// TIA Portal V17 export
// export: Created 2022-02-08T17:35:46.0434101Z, ExportSetting WithDefaults, DisplayName Totally Integrated Automation Portal, DisplayVersion V17 Update 2, DisplayName TIA Portal Openness, DisplayVersion V17 Update 2, DisplayName TIA Portal Version Control Interface, DisplayVersion V17, DisplayName STEP 7 Professional, DisplayVersion V17 Update 2, DisplayName STEP 7 Safety, DisplayVersion V17, DisplayName WinCC UA Professional, DisplayVersion V17 Update 2
FUNCTION_BLOCK "Motor"   // FB2, FBD
TITLE = Control module: Motor
{ S7_Optimized_Access := 'TRUE' }
VERSION : 0.1
// stored: AutoNumber true, IsIECCheckEnabled false, IsRetainMemResEnabled false, MemoryReserve 100, SetENOAutomatically false, UDAEnableTagReadback false
   VAR_INPUT
      i_Thermal : Bool;
      i_Mainswitch : Bool;
      i_SpareAlarm1 : Bool;
      i_SpareAlarm2 : Bool;
      i_SpareAlarm3 : Bool;
      i_SpareAlarm4 : Bool;
      i_InterlockDir1 : Bool;
      i_InterlockDir2 : Bool;
      i_EndswitchDir1 : Bool;
      i_EndswitchDir2 : Bool;
   END_VAR
   VAR_OUTPUT
      q_Dir1 : Bool;
      q_Dir2 : Bool;
      q_HighSpeed : Bool;
   END_VAR
   VAR_IN_OUT
      PLC_CtrlMod : "PLC_CtrlMod";
      HMI_CtrlMod : "HMI_CtrlMod";
   END_VAR
   VAR
      s_ManualMode : Bool;
      s_AutomaticMode : Bool;
      s_Direction1 : Bool;
      s_Direction2 : Bool;
      s_Alarms : Struct
         ThermalFaults : Bool;
         MainswitchOff : Bool;
         SpareAlarm1 : Bool;
         SpareAlarm2 : Bool;
         SpareAlarm3 : Bool;
         SpareAlarm4 : Bool;
      END_STRUCT;
   END_VAR
BEGIN

REGION Network 1: Selection manual mode
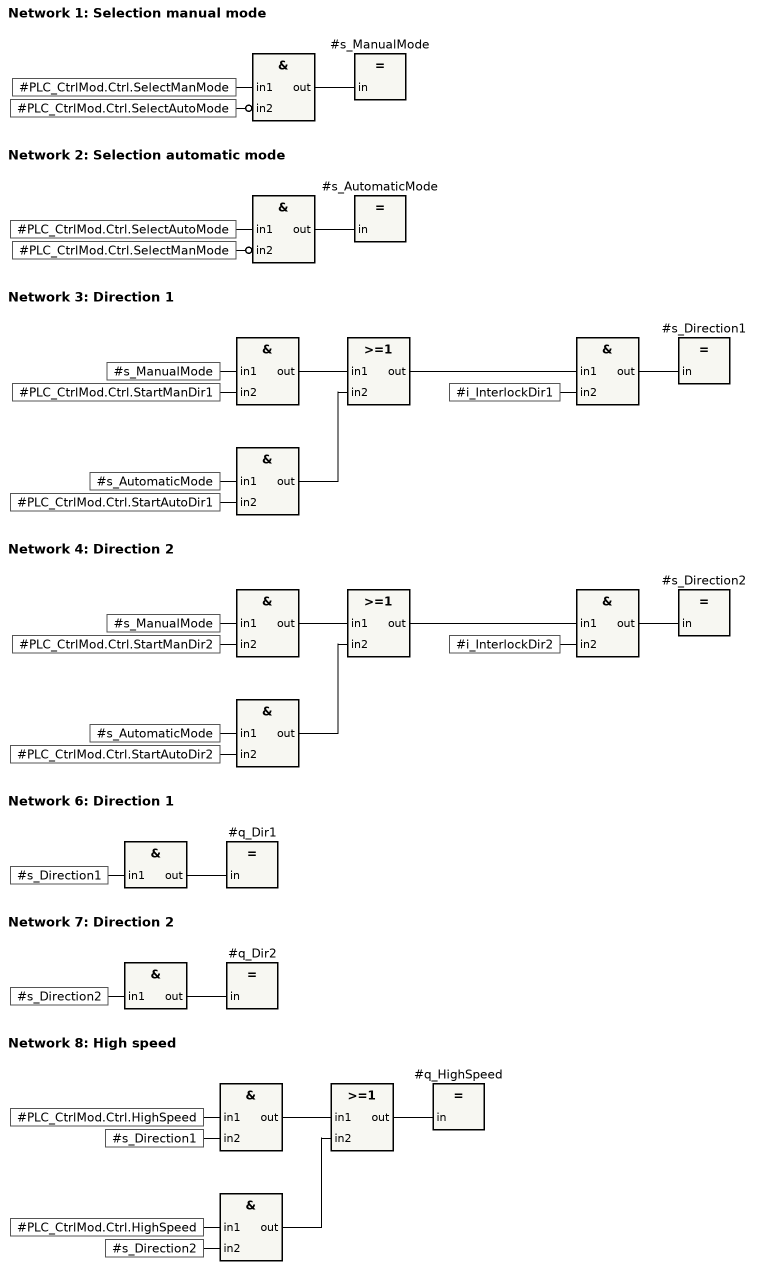
   #s_ManualMode := #PLC_CtrlMod.Ctrl.SelectManMode AND NOT #PLC_CtrlMod.Ctrl.SelectAutoMode;
END_REGION

REGION Network 2: Selection automatic mode
   #s_AutomaticMode := #PLC_CtrlMod.Ctrl.SelectAutoMode AND NOT #PLC_CtrlMod.Ctrl.SelectManMode;
END_REGION

REGION Network 3: Direction 1
   #s_Direction1 := ((#s_ManualMode AND #PLC_CtrlMod.Ctrl.StartManDir1) OR (#s_AutomaticMode AND #PLC_CtrlMod.Ctrl.StartAutoDir1)) AND #i_InterlockDir1;
END_REGION

REGION Network 4: Direction 2
   #s_Direction2 := ((#s_ManualMode AND #PLC_CtrlMod.Ctrl.StartManDir2) OR (#s_AutomaticMode AND #PLC_CtrlMod.Ctrl.StartAutoDir2)) AND #i_InterlockDir2;
END_REGION

REGION Network 5: ********* OUTPUTS *********
END_REGION

REGION Network 6: Direction 1
   #q_Dir1 := #s_Direction1;
END_REGION

REGION Network 7: Direction 2
   #q_Dir2 := #s_Direction2;
END_REGION

REGION Network 8: High speed
   #q_HighSpeed := (#PLC_CtrlMod.Ctrl.HighSpeed AND #s_Direction1) OR (#PLC_CtrlMod.Ctrl.HighSpeed AND #s_Direction2);
END_REGION

REGION Network 9: ********* ALARMS *********
END_REGION

REGION Network 10: Thermal fault
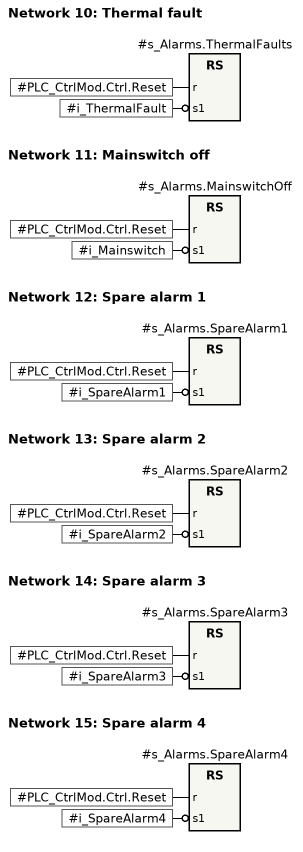
   IF #PLC_CtrlMod.Ctrl.Reset THEN
       #s_Alarms.ThermalFaults := FALSE;   // RS flip-flop
   END_IF;
   IF NOT #i_ThermalFault THEN #s_Alarms.ThermalFaults := TRUE; END_IF;
END_REGION

REGION Network 11: Mainswitch off
   IF #PLC_CtrlMod.Ctrl.Reset THEN
       #s_Alarms.MainswitchOff := FALSE;   // RS flip-flop
   END_IF;
   IF NOT #i_Mainswitch THEN #s_Alarms.MainswitchOff := TRUE; END_IF;
END_REGION

REGION Network 12: Spare alarm 1
   IF #PLC_CtrlMod.Ctrl.Reset THEN
       #s_Alarms.SpareAlarm1 := FALSE;   // RS flip-flop
   END_IF;
   IF NOT #i_SpareAlarm1 THEN #s_Alarms.SpareAlarm1 := TRUE; END_IF;
END_REGION

REGION Network 13: Spare alarm 2
   IF #PLC_CtrlMod.Ctrl.Reset THEN
       #s_Alarms.SpareAlarm2 := FALSE;   // RS flip-flop
   END_IF;
   IF NOT #i_SpareAlarm2 THEN #s_Alarms.SpareAlarm2 := TRUE; END_IF;
END_REGION

REGION Network 14: Spare alarm 3
   IF #PLC_CtrlMod.Ctrl.Reset THEN
       #s_Alarms.SpareAlarm3 := FALSE;   // RS flip-flop
   END_IF;
   IF NOT #i_SpareAlarm3 THEN #s_Alarms.SpareAlarm3 := TRUE; END_IF;
END_REGION

REGION Network 15: Spare alarm 4
   IF #PLC_CtrlMod.Ctrl.Reset THEN
       #s_Alarms.SpareAlarm4 := FALSE;   // RS flip-flop
   END_IF;
   IF NOT #i_SpareAlarm4 THEN #s_Alarms.SpareAlarm4 := TRUE; END_IF;
END_REGION
END_FUNCTION_BLOCK
